PROGRAM MANIPULATOR
VAR
	_context : fbManipulatorContext;
END_VAR

_context.Run();

END_PROGRAM

(* stored: Version 1.1.0.1, ProductVersion 3.1.4024.6
   POU MANIPULATOR: Id {46649b69-6523-450e-95e7-0d33168f6b81}, SpecialFunc None *)
